{attribute 'qualified_only'}
VAR_GLOBAL
	AX_StructModbusTCP 	AT %MW112 	: ARRAY[1..10000] OF WORD;
END_VAR

(* stored: Version 1.1.0.1, ProductVersion 3.1.4024.9
   GVL GVL_DataBaseStructures: Id {38e58985-13d8-4d54-aae1-0c5e77824ddf} *)
